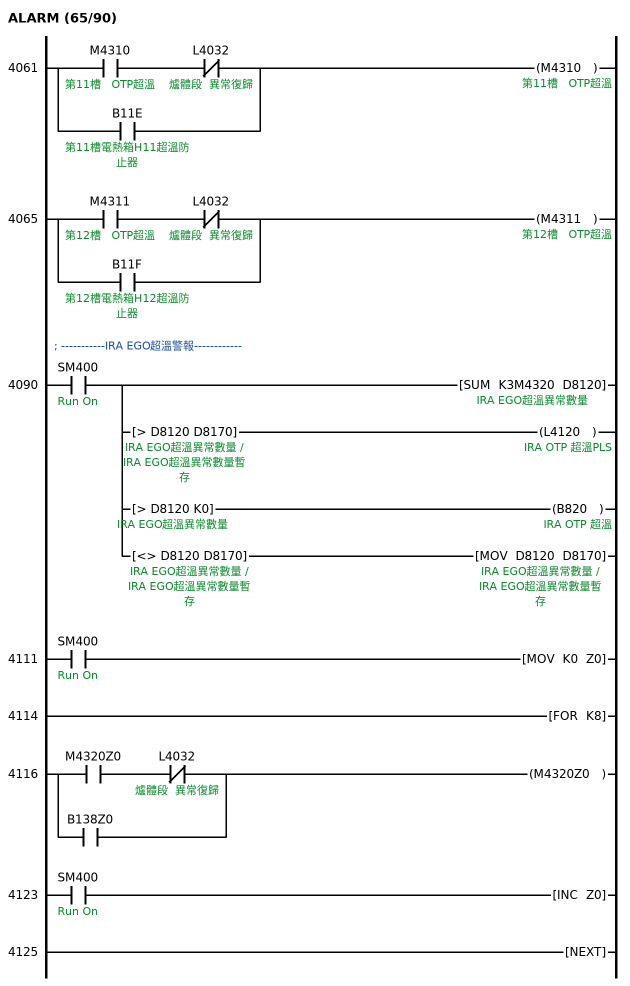
[picture p240: ladder of ALARM, rungs at steps 4061 to 4125]
4061  LD      M4310  ; 第11槽   OTP超溫
      ANI     L4032  ; 爐體段  異常復歸
      OR      B11E  ; 第11槽電熱箱H11超溫防止器
      OUT     M4310  ; 第11槽   OTP超溫
4065  LD      M4311  ; 第12槽   OTP超溫
      ANI     L4032  ; 爐體段  異常復歸
      OR      B11F  ; 第12槽電熱箱H12超溫防止器
      OUT     M4311  ; 第12槽   OTP超溫
; -----------IRA EGO超溫警報------------
4090  LD      SM400  ; Run On
      SUM     K3M4320 D8120  ; 第01槽  IRA OTP 超溫 / IRA EGO超溫異常數量
      MPS
      AND>    D8120 D8170  ; IRA EGO超溫異常數量 / IRA EGO超溫異常數量暫存
      OUT     L4120  ; IRA OTP 超溫PLS
      MRD
      AND>    D8120 K0  ; IRA EGO超溫異常數量
      OUT     B820  ; IRA OTP 超溫
      MPP
      AND<>   D8120 D8170  ; IRA EGO超溫異常數量 / IRA EGO超溫異常數量暫存
      MOV     D8120 D8170
4111  LD      SM400  ; Run On
      MOV     K0 Z0
4114  FOR     K8
4116  LD      M4320Z0
      ANI     L4032  ; 爐體段  異常復歸
      OR      B138Z0
      OUT     M4320Z0
4123  LD      SM400  ; Run On
      INC     Z0
4125  NEXT
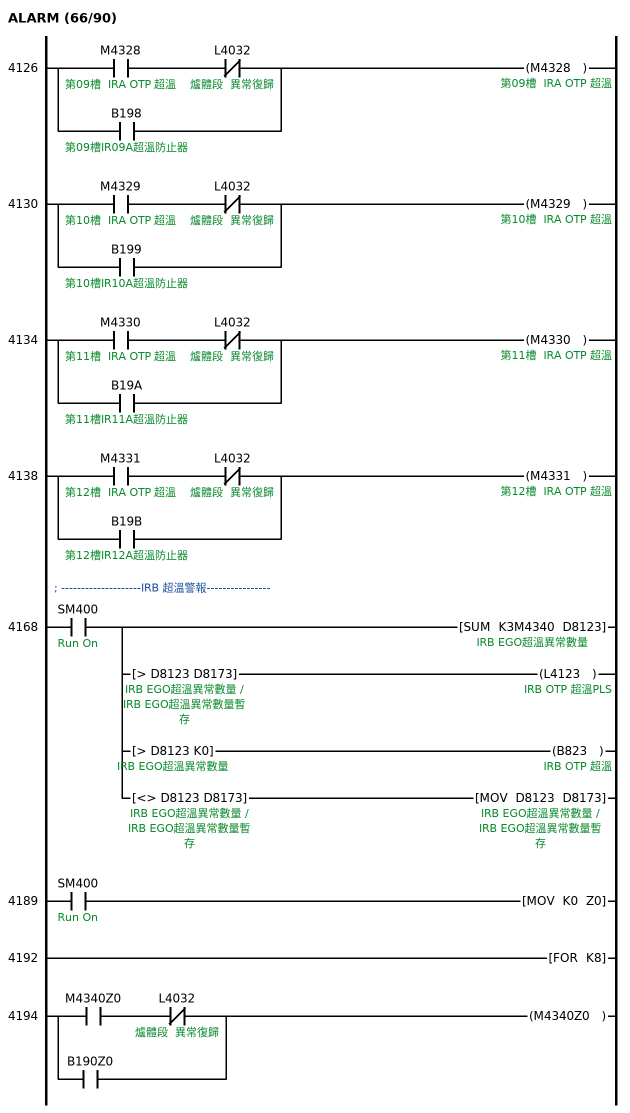
4126  LD      M4328  ; 第09槽  IRA OTP 超溫
      ANI     L4032  ; 爐體段  異常復歸
      OR      B198  ; 第09槽IR09A超溫防止器
      OUT     M4328  ; 第09槽  IRA OTP 超溫
4130  LD      M4329  ; 第10槽  IRA OTP 超溫
      ANI     L4032  ; 爐體段  異常復歸
      OR      B199  ; 第10槽IR10A超溫防止器
      OUT     M4329  ; 第10槽  IRA OTP 超溫
4134  LD      M4330  ; 第11槽  IRA OTP 超溫
      ANI     L4032  ; 爐體段  異常復歸
      OR      B19A  ; 第11槽IR11A超溫防止器
      OUT     M4330  ; 第11槽  IRA OTP 超溫
4138  LD      M4331  ; 第12槽  IRA OTP 超溫
      ANI     L4032  ; 爐體段  異常復歸
      OR      B19B  ; 第12槽IR12A超溫防止器
      OUT     M4331  ; 第12槽  IRA OTP 超溫
; --------------------IRB 超溫警報----------------
4168  LD      SM400  ; Run On
      SUM     K3M4340 D8123  ; 第01槽  IRB OTP 超溫 / IRB EGO超溫異常數量
      MPS
      AND>    D8123 D8173  ; IRB EGO超溫異常數量 / IRB EGO超溫異常數量暫存
      OUT     L4123  ; IRB OTP 超溫PLS
      MRD
      AND>    D8123 K0  ; IRB EGO超溫異常數量
      OUT     B823  ; IRB OTP 超溫
      MPP
      AND<>   D8123 D8173  ; IRB EGO超溫異常數量 / IRB EGO超溫異常數量暫存
      MOV     D8123 D8173
4189  LD      SM400  ; Run On
      MOV     K0 Z0
4192  FOR     K8
4194  LD      M4340Z0
      ANI     L4032  ; 爐體段  異常復歸
      OR      B190Z0
      OUT     M4340Z0
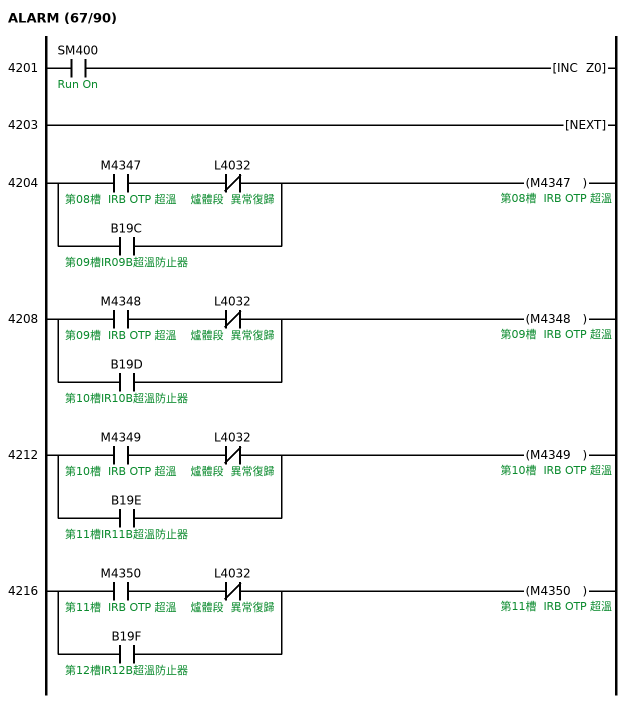
4201  LD      SM400  ; Run On
      INC     Z0
4203  NEXT
4204  LD      M4347  ; 第08槽  IRB OTP 超溫
      ANI     L4032  ; 爐體段  異常復歸
      OR      B19C  ; 第09槽IR09B超溫防止器
      OUT     M4347  ; 第08槽  IRB OTP 超溫
4208  LD      M4348  ; 第09槽  IRB OTP 超溫
      ANI     L4032  ; 爐體段  異常復歸
      OR      B19D  ; 第10槽IR10B超溫防止器
      OUT     M4348  ; 第09槽  IRB OTP 超溫
4212  LD      M4349  ; 第10槽  IRB OTP 超溫
      ANI     L4032  ; 爐體段  異常復歸
      OR      B19E  ; 第11槽IR11B超溫防止器
      OUT     M4349  ; 第10槽  IRB OTP 超溫
4216  LD      M4350  ; 第11槽  IRB OTP 超溫
      ANI     L4032  ; 爐體段  異常復歸
      OR      B19F  ; 第12槽IR12B超溫防止器
      OUT     M4350  ; 第11槽  IRB OTP 超溫
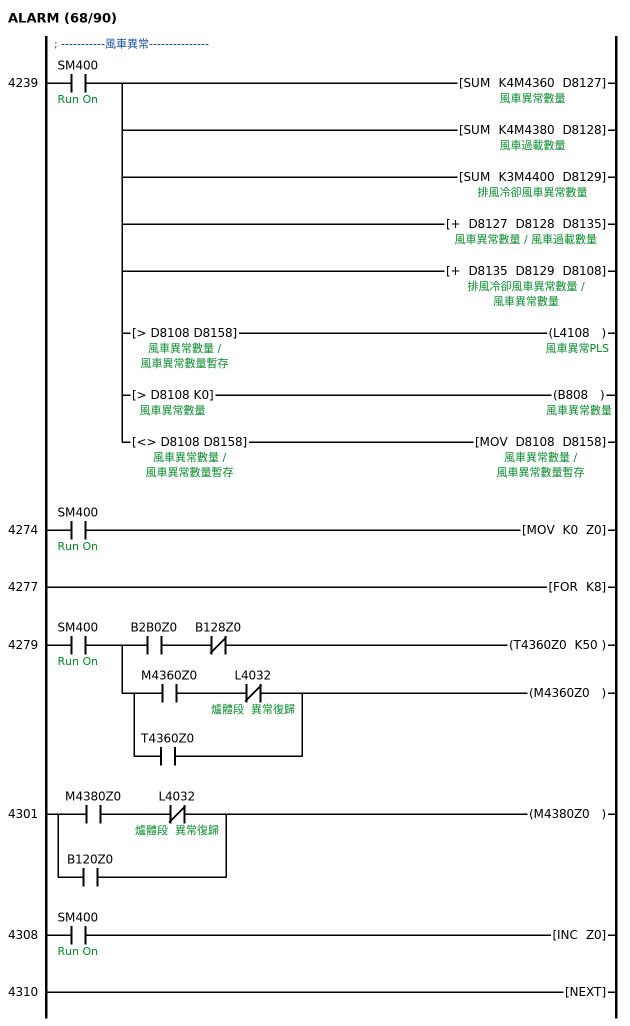
; -----------風車異常---------------
4239  LD      SM400  ; Run On
      SUM     K4M4360 D8127  ; 第01槽  風車馬達異常 / 風車異常數量
      SUM     K4M4380 D8128  ; 第01槽  風車馬達過載 / 風車過載數量
      SUM     K3M4400 D8129  ; 進料輸送排氣風車異常 / 排風冷卻風車異常數量
      +       D8127 D8128 D8135
      +       D8135 D8129 D8108  ; 風車異常數量
      MPS
      AND>    D8108 D8158  ; 風車異常數量 / 風車異常數量暫存
      OUT     L4108  ; 風車異常PLS
      MRD
      AND>    D8108 K0  ; 風車異常數量
      OUT     B808  ; 風車異常數量
      MPP
      AND<>   D8108 D8158  ; 風車異常數量 / 風車異常數量暫存
      MOV     D8108 D8158
4274  LD      SM400  ; Run On
      MOV     K0 Z0
4277  FOR     K8
4279  LD      SM400  ; Run On
      MPS
      AND     B2B0Z0
      ANI     B128Z0
      OUT     T4360Z0 K50
      MPP
      LD      M4360Z0
      ANI     L4032  ; 爐體段  異常復歸
      OR      T4360Z0
      ANB
      OUT     M4360Z0
4301  LD      M4380Z0
      ANI     L4032  ; 爐體段  異常復歸
      OR      B120Z0
      OUT     M4380Z0
4308  LD      SM400  ; Run On
      INC     Z0
4310  NEXT
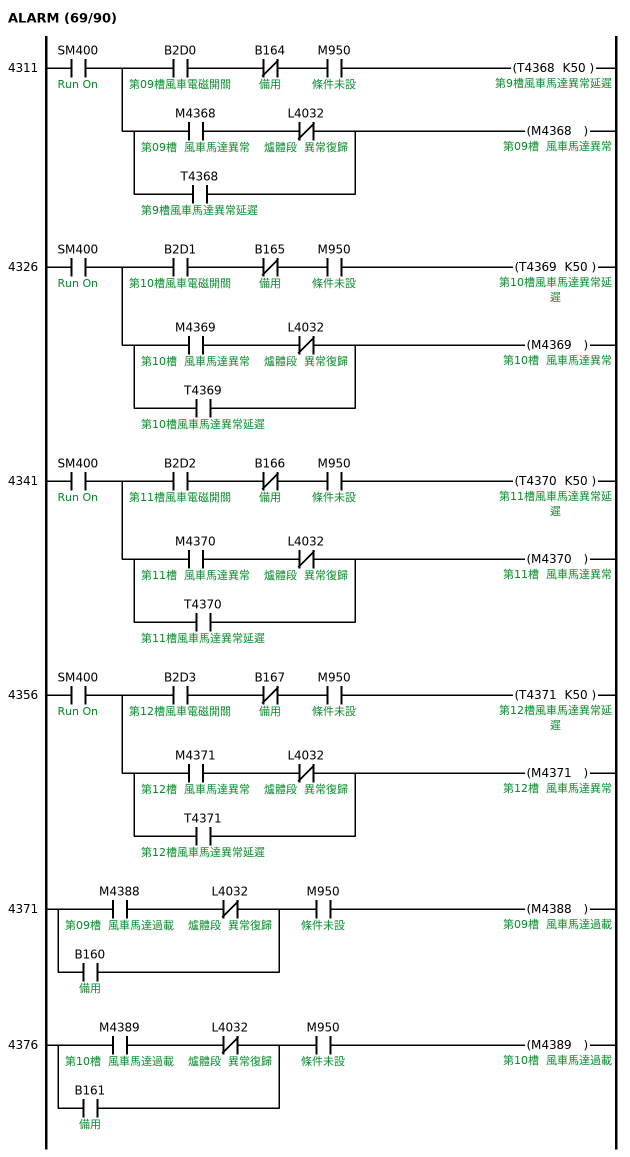
4311  LD      SM400  ; Run On
      MPS
      AND     B2D0  ; 第09槽風車電磁開關
      ANI     B164  ; 備用
      AND     M950  ; 條件未設
      OUT     T4368 K50  ; 第9槽風車馬達異常延遲
      MPP
      LD      M4368  ; 第09槽  風車馬達異常
      ANI     L4032  ; 爐體段  異常復歸
      OR      T4368  ; 第9槽風車馬達異常延遲
      ANB
      OUT     M4368  ; 第09槽  風車馬達異常
4326  LD      SM400  ; Run On
      MPS
      AND     B2D1  ; 第10槽風車電磁開關
      ANI     B165  ; 備用
      AND     M950  ; 條件未設
      OUT     T4369 K50  ; 第10槽風車馬達異常延遲
      MPP
      LD      M4369  ; 第10槽  風車馬達異常
      ANI     L4032  ; 爐體段  異常復歸
      OR      T4369  ; 第10槽風車馬達異常延遲
      ANB
      OUT     M4369  ; 第10槽  風車馬達異常
4341  LD      SM400  ; Run On
      MPS
      AND     B2D2  ; 第11槽風車電磁開關
      ANI     B166  ; 備用
      AND     M950  ; 條件未設
      OUT     T4370 K50  ; 第11槽風車馬達異常延遲
      MPP
      LD      M4370  ; 第11槽  風車馬達異常
      ANI     L4032  ; 爐體段  異常復歸
      OR      T4370  ; 第11槽風車馬達異常延遲
      ANB
      OUT     M4370  ; 第11槽  風車馬達異常
4356  LD      SM400  ; Run On
      MPS
      AND     B2D3  ; 第12槽風車電磁開關
      ANI     B167  ; 備用
      AND     M950  ; 條件未設
      OUT     T4371 K50  ; 第12槽風車馬達異常延遲
      MPP
      LD      M4371  ; 第12槽  風車馬達異常
      ANI     L4032  ; 爐體段  異常復歸
      OR      T4371  ; 第12槽風車馬達異常延遲
      ANB
      OUT     M4371  ; 第12槽  風車馬達異常
4371  LD      M4388  ; 第09槽  風車馬達過載
      ANI     L4032  ; 爐體段  異常復歸
      OR      B160  ; 備用
      AND     M950  ; 條件未設
      OUT     M4388  ; 第09槽  風車馬達過載
4376  LD      M4389  ; 第10槽  風車馬達過載
      ANI     L4032  ; 爐體段  異常復歸
      OR      B161  ; 備用
      AND     M950  ; 條件未設
      OUT     M4389  ; 第10槽  風車馬達過載
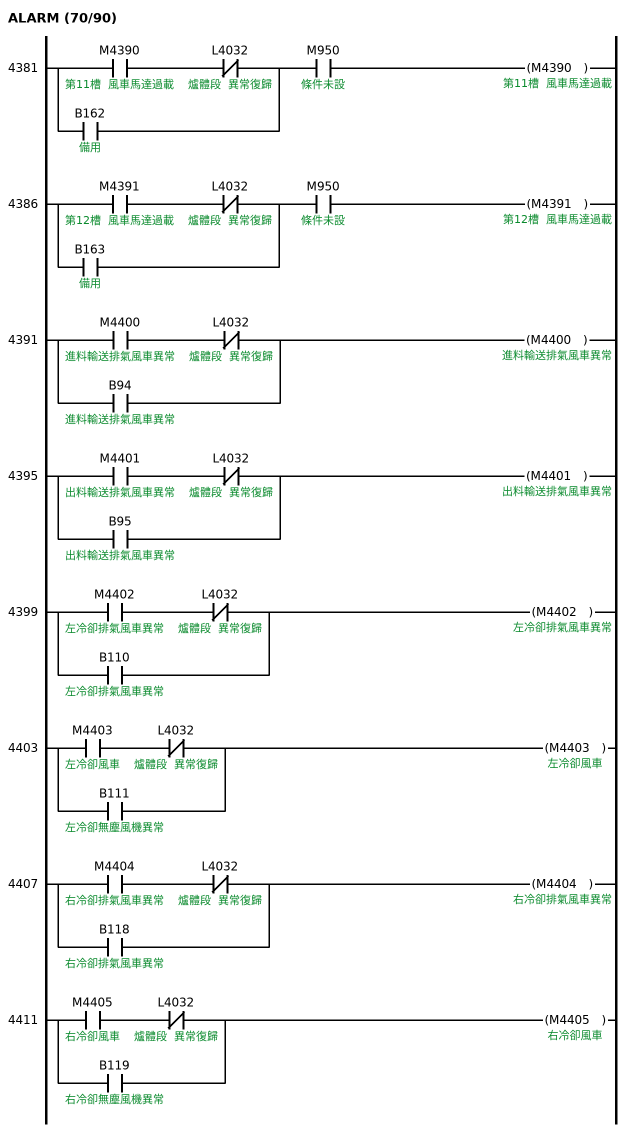
4381  LD      M4390  ; 第11槽  風車馬達過載
      ANI     L4032  ; 爐體段  異常復歸
      OR      B162  ; 備用
      AND     M950  ; 條件未設
      OUT     M4390  ; 第11槽  風車馬達過載
4386  LD      M4391  ; 第12槽  風車馬達過載
      ANI     L4032  ; 爐體段  異常復歸
      OR      B163  ; 備用
      AND     M950  ; 條件未設
      OUT     M4391  ; 第12槽  風車馬達過載
4391  LD      M4400  ; 進料輸送排氣風車異常
      ANI     L4032  ; 爐體段  異常復歸
      OR      B94  ; 進料輸送排氣風車異常
      OUT     M4400  ; 進料輸送排氣風車異常
4395  LD      M4401  ; 出料輸送排氣風車異常
      ANI     L4032  ; 爐體段  異常復歸
      OR      B95  ; 出料輸送排氣風車異常
      OUT     M4401  ; 出料輸送排氣風車異常
4399  LD      M4402  ; 左冷卻排氣風車異常
      ANI     L4032  ; 爐體段  異常復歸
      OR      B110  ; 左冷卻排氣風車異常
      OUT     M4402  ; 左冷卻排氣風車異常
4403  LD      M4403  ; 左冷卻風車
      ANI     L4032  ; 爐體段  異常復歸
      OR      B111  ; 左冷卻無塵風機異常
      OUT     M4403  ; 左冷卻風車
4407  LD      M4404  ; 右冷卻排氣風車異常
      ANI     L4032  ; 爐體段  異常復歸
      OR      B118  ; 右冷卻排氣風車異常
      OUT     M4404  ; 右冷卻排氣風車異常
4411  LD      M4405  ; 右冷卻風車
      ANI     L4032  ; 爐體段  異常復歸
      OR      B119  ; 右冷卻無塵風機異常
      OUT     M4405  ; 右冷卻風車
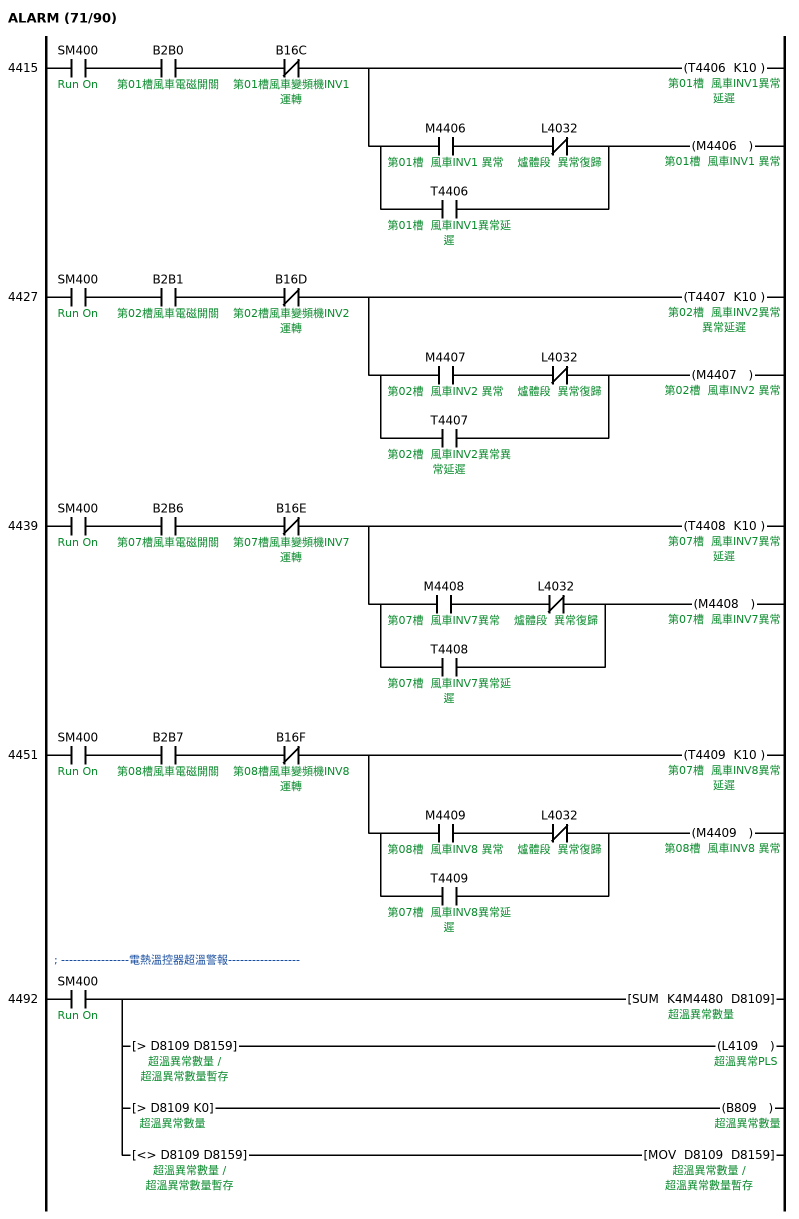
4415  LD      SM400  ; Run On
      AND     B2B0  ; 第01槽風車電磁開關
      ANI     B16C  ; 第01槽風車變頻機INV1運轉
      OUT     T4406 K10  ; 第01槽  風車INV1異常延遲
      LD      M4406  ; 第01槽  風車INV1 異常
      ANI     L4032  ; 爐體段  異常復歸
      OR      T4406  ; 第01槽  風車INV1異常延遲
      ANB
      OUT     M4406  ; 第01槽  風車INV1 異常
4427  LD      SM400  ; Run On
      AND     B2B1  ; 第02槽風車電磁開關
      ANI     B16D  ; 第02槽風車變頻機INV2運轉
      OUT     T4407 K10  ; 第02槽  風車INV2異常異常延遲
      LD      M4407  ; 第02槽  風車INV2 異常
      ANI     L4032  ; 爐體段  異常復歸
      OR      T4407  ; 第02槽  風車INV2異常異常延遲
      ANB
      OUT     M4407  ; 第02槽  風車INV2 異常
4439  LD      SM400  ; Run On
      AND     B2B6  ; 第07槽風車電磁開關
      ANI     B16E  ; 第07槽風車變頻機INV7運轉
      OUT     T4408 K10  ; 第07槽  風車INV7異常延遲
      LD      M4408  ; 第07槽  風車INV7異常
      ANI     L4032  ; 爐體段  異常復歸
      OR      T4408  ; 第07槽  風車INV7異常延遲
      ANB
      OUT     M4408  ; 第07槽  風車INV7異常
4451  LD      SM400  ; Run On
      AND     B2B7  ; 第08槽風車電磁開關
      ANI     B16F  ; 第08槽風車變頻機INV8運轉
      OUT     T4409 K10  ; 第07槽  風車INV8異常延遲
      LD      M4409  ; 第08槽  風車INV8 異常
      ANI     L4032  ; 爐體段  異常復歸
      OR      T4409  ; 第07槽  風車INV8異常延遲
      ANB
      OUT     M4409  ; 第08槽  風車INV8 異常
; -----------------電熱溫控器超溫警報------------------
4492  LD      SM400  ; Run On
      SUM     K4M4480 D8109  ; 第01槽 熱風超溫異常 / 超溫異常數量
      MPS
      AND>    D8109 D8159  ; 超溫異常數量 / 超溫異常數量暫存
      OUT     L4109  ; 超溫異常PLS
      MRD
      AND>    D8109 K0  ; 超溫異常數量
      OUT     B809  ; 超溫異常數量
      MPP
      AND<>   D8109 D8159  ; 超溫異常數量 / 超溫異常數量暫存
      MOV     D8109 D8159
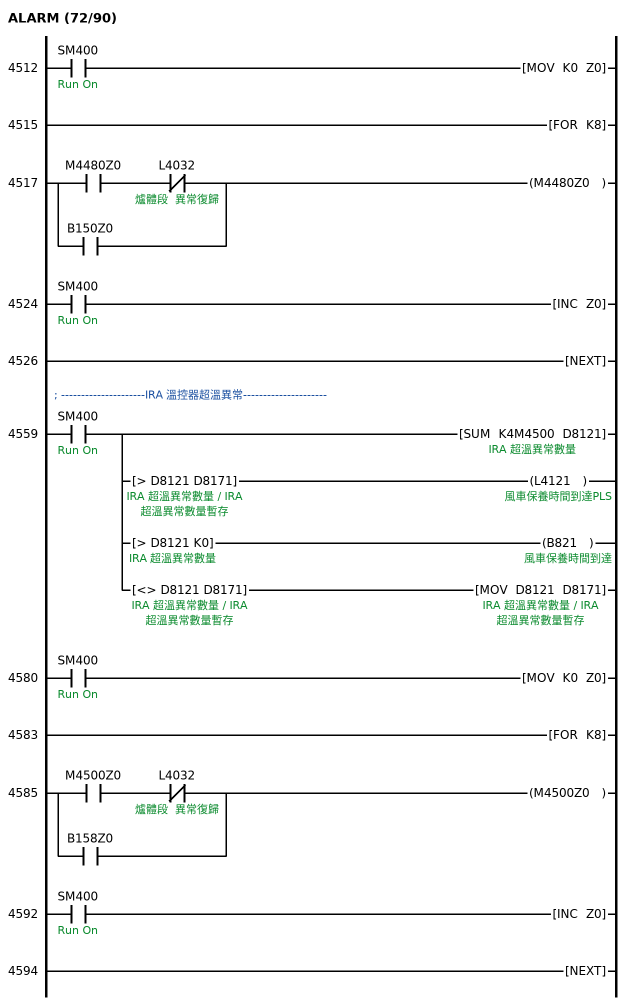
4512  LD      SM400  ; Run On
      MOV     K0 Z0
4515  FOR     K8
4517  LD      M4480Z0
      ANI     L4032  ; 爐體段  異常復歸
      OR      B150Z0
      OUT     M4480Z0
4524  LD      SM400  ; Run On
      INC     Z0
4526  NEXT
; ---------------------IRA 溫控器超溫異常---------------------
4559  LD      SM400  ; Run On
      SUM     K4M4500 D8121  ; 第1槽 IRA 超溫異常 / IRA 超溫異常數量
      MPS
      AND>    D8121 D8171  ; IRA 超溫異常數量 / IRA 超溫異常數量暫存
      OUT     L4121  ; 風車保養時間到達PLS
      MRD
      AND>    D8121 K0  ; IRA 超溫異常數量
      OUT     B821  ; 風車保養時間到達
      MPP
      AND<>   D8121 D8171  ; IRA 超溫異常數量 / IRA 超溫異常數量暫存
      MOV     D8121 D8171
4580  LD      SM400  ; Run On
      MOV     K0 Z0
4583  FOR     K8
4585  LD      M4500Z0
      ANI     L4032  ; 爐體段  異常復歸
      OR      B158Z0
      OUT     M4500Z0
4592  LD      SM400  ; Run On
      INC     Z0
4594  NEXT
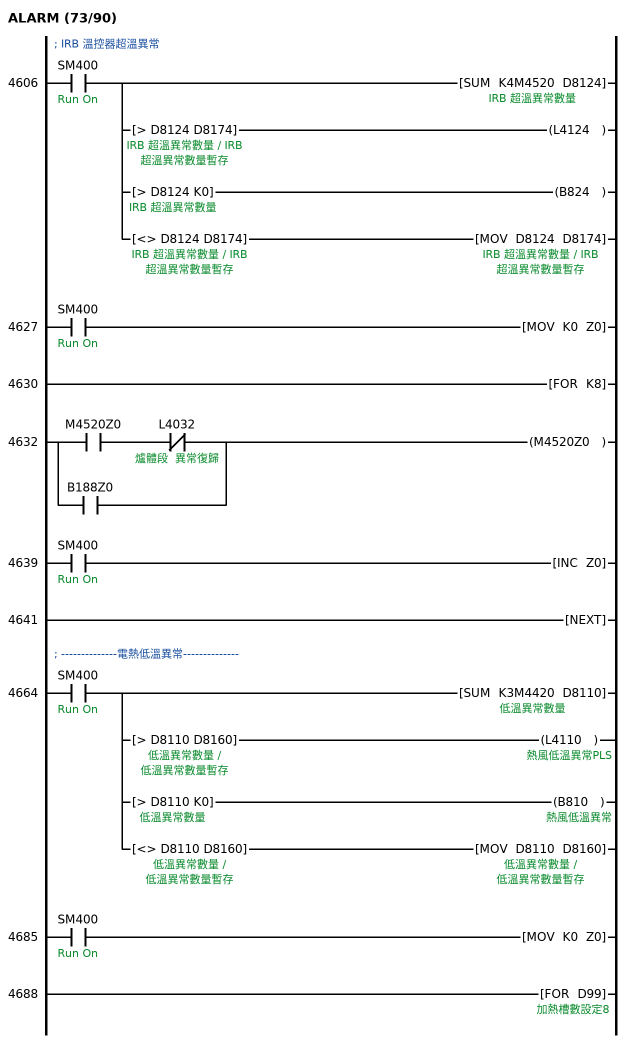
; IRB 溫控器超溫異常
4606  LD      SM400  ; Run On
      SUM     K4M4520 D8124  ; 第1槽 IRB 超溫異常 / IRB 超溫異常數量
      MPS
      AND>    D8124 D8174  ; IRB 超溫異常數量 / IRB 超溫異常數量暫存
      OUT     L4124
      MRD
      AND>    D8124 K0  ; IRB 超溫異常數量
      OUT     B824
      MPP
      AND<>   D8124 D8174  ; IRB 超溫異常數量 / IRB 超溫異常數量暫存
      MOV     D8124 D8174
4627  LD      SM400  ; Run On
      MOV     K0 Z0
4630  FOR     K8
4632  LD      M4520Z0
      ANI     L4032  ; 爐體段  異常復歸
      OR      B188Z0
      OUT     M4520Z0
4639  LD      SM400  ; Run On
      INC     Z0
4641  NEXT
; --------------電熱低溫異常--------------
4664  LD      SM400  ; Run On
      SUM     K3M4420 D8110  ; 第01槽 熱風低溫異常 / 低溫異常數量
      MPS
      AND>    D8110 D8160  ; 低溫異常數量 / 低溫異常數量暫存
      OUT     L4110  ; 熱風低溫異常PLS
      MRD
      AND>    D8110 K0  ; 低溫異常數量
      OUT     B810  ; 熱風低溫異常
      MPP
      AND<>   D8110 D8160  ; 低溫異常數量 / 低溫異常數量暫存
      MOV     D8110 D8160
4685  LD      SM400  ; Run On
      MOV     K0 Z0
4688  FOR     D99  ; 加熱槽數設定8
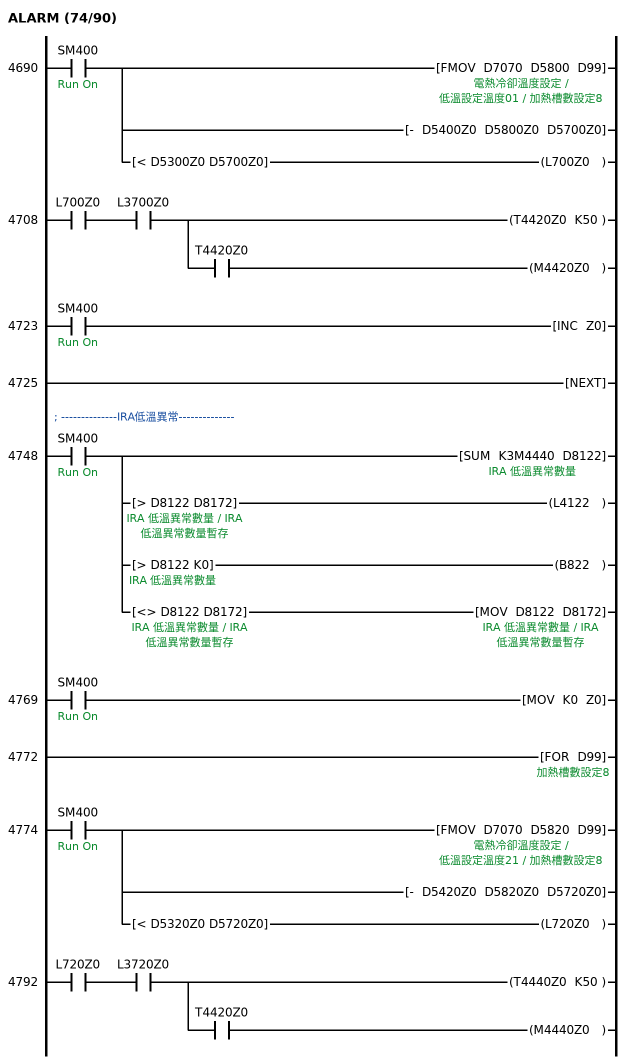
4690  LD      SM400  ; Run On
      FMOV    D7070 D5800 D99  ; 電熱冷卻溫度設定 / 低溫設定溫度01
      -       D5400Z0 D5800Z0 D5700Z0
      AND<    D5300Z0 D5700Z0
      OUT     L700Z0
4708  LD      L700Z0
      AND     L3700Z0
      OUT     T4420Z0 K50
      AND     T4420Z0
      OUT     M4420Z0
4723  LD      SM400  ; Run On
      INC     Z0
4725  NEXT
; --------------IRA低溫異常--------------
4748  LD      SM400  ; Run On
      SUM     K3M4440 D8122  ; 第01槽 IRA 低溫異常 / IRA 低溫異常數量
      MPS
      AND>    D8122 D8172  ; IRA 低溫異常數量 / IRA 低溫異常數量暫存
      OUT     L4122
      MRD
      AND>    D8122 K0  ; IRA 低溫異常數量
      OUT     B822
      MPP
      AND<>   D8122 D8172  ; IRA 低溫異常數量 / IRA 低溫異常數量暫存
      MOV     D8122 D8172
4769  LD      SM400  ; Run On
      MOV     K0 Z0
4772  FOR     D99
4774  LD      SM400  ; Run On
      FMOV    D7070 D5820 D99  ; 低溫設定溫度21
      -       D5420Z0 D5820Z0 D5720Z0
      AND<    D5320Z0 D5720Z0
      OUT     L720Z0
4792  LD      L720Z0
      AND     L3720Z0
      OUT     T4440Z0 K50
      AND     T4420Z0
      OUT     M4440Z0
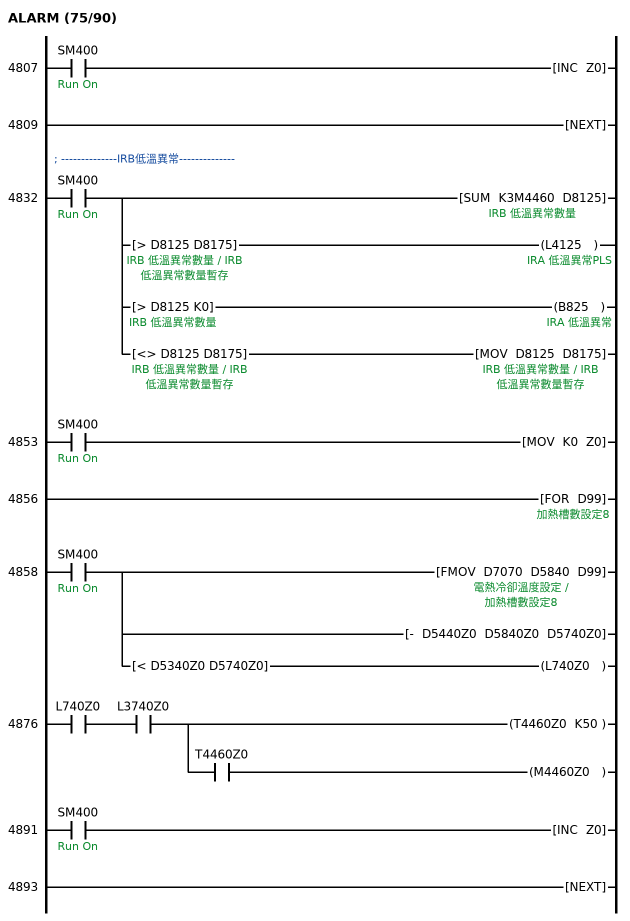
4807  LD      SM400  ; Run On
      INC     Z0
4809  NEXT
; --------------IRB低溫異常--------------
4832  LD      SM400  ; Run On
      SUM     K3M4460 D8125  ; 第01槽 IRB 低溫異常 / IRB 低溫異常數量
      MPS
      AND>    D8125 D8175  ; IRB 低溫異常數量 / IRB 低溫異常數量暫存
      OUT     L4125  ; IRA 低溫異常PLS
      MRD
      AND>    D8125 K0  ; IRB 低溫異常數量
      OUT     B825  ; IRA 低溫異常
      MPP
      AND<>   D8125 D8175  ; IRB 低溫異常數量 / IRB 低溫異常數量暫存
      MOV     D8125 D8175
4853  LD      SM400  ; Run On
      MOV     K0 Z0
4856  FOR     D99
4858  LD      SM400  ; Run On
      FMOV    D7070 D5840 D99
      -       D5440Z0 D5840Z0 D5740Z0
      AND<    D5340Z0 D5740Z0
      OUT     L740Z0
4876  LD      L740Z0
      AND     L3740Z0
      OUT     T4460Z0 K50
      AND     T4460Z0
      OUT     M4460Z0
4891  LD      SM400  ; Run On
      INC     Z0
4893  NEXT
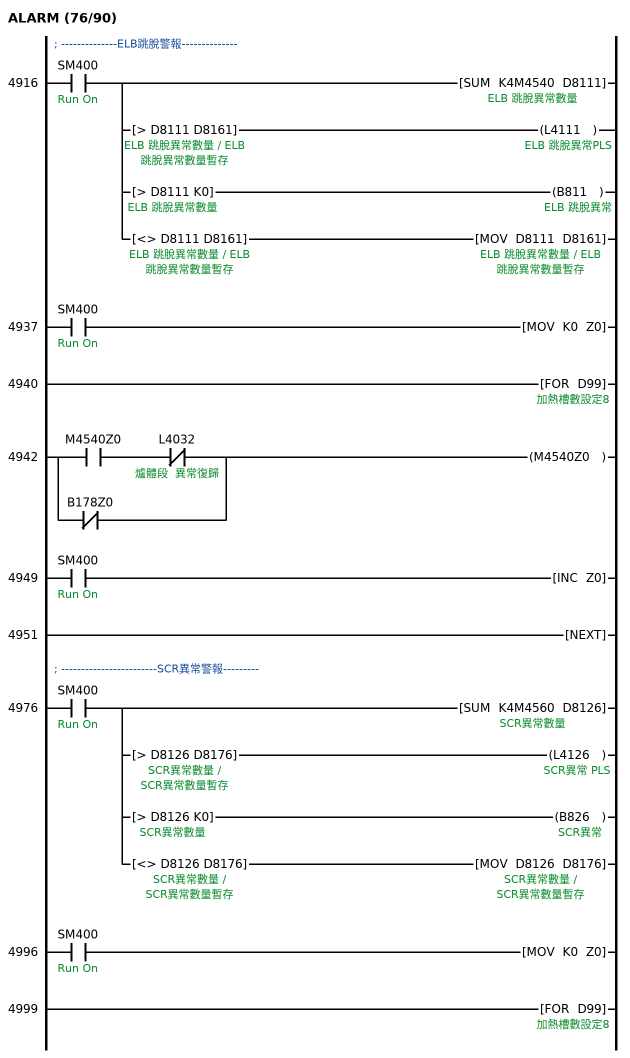
; --------------ELB跳脫警報--------------
4916  LD      SM400  ; Run On
      SUM     K4M4540 D8111  ; 第01槽  分路開關跳脫異常 / ELB 跳脫異常數量
      MPS
      AND>    D8111 D8161  ; ELB 跳脫異常數量 / ELB 跳脫異常數量暫存
      OUT     L4111  ; ELB 跳脫異常PLS
      MRD
      AND>    D8111 K0  ; ELB 跳脫異常數量
      OUT     B811  ; ELB 跳脫異常
      MPP
      AND<>   D8111 D8161  ; ELB 跳脫異常數量 / ELB 跳脫異常數量暫存
      MOV     D8111 D8161
4937  LD      SM400  ; Run On
      MOV     K0 Z0
4940  FOR     D99
4942  LD      M4540Z0
      ANI     L4032  ; 爐體段  異常復歸
      ORI     B178Z0
      OUT     M4540Z0
4949  LD      SM400  ; Run On
      INC     Z0
4951  NEXT
; ------------------------SCR異常警報---------
4976  LD      SM400  ; Run On
      SUM     K4M4560 D8126  ; 第01槽  SCR異常 / SCR異常數量
      MPS
      AND>    D8126 D8176  ; SCR異常數量 / SCR異常數量暫存
      OUT     L4126  ; SCR異常 PLS
      MRD
      AND>    D8126 K0  ; SCR異常數量
      OUT     B826  ; SCR異常
      MPP
      AND<>   D8126 D8176  ; SCR異常數量 / SCR異常數量暫存
      MOV     D8126 D8176
4996  LD      SM400  ; Run On
      MOV     K0 Z0
4999  FOR     D99
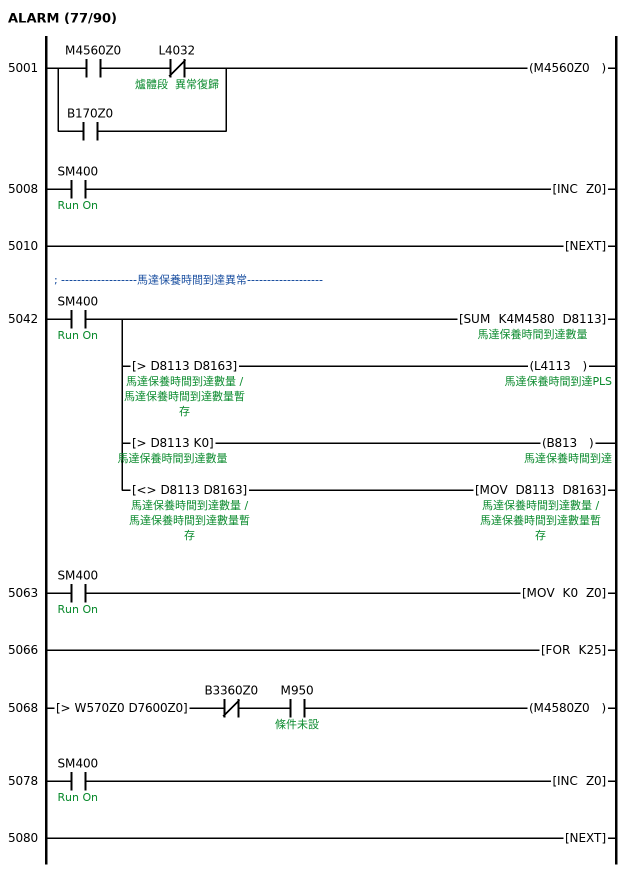
5001  LD      M4560Z0
      ANI     L4032  ; 爐體段  異常復歸
      OR      B170Z0
      OUT     M4560Z0
5008  LD      SM400  ; Run On
      INC     Z0
5010  NEXT
; -------------------馬達保養時間到達異常-------------------
5042  LD      SM400  ; Run On
      SUM     K4M4580 D8113  ; 馬達保養時間到達數量
      MPS
      AND>    D8113 D8163  ; 馬達保養時間到達數量 / 馬達保養時間到達數量暫存
      OUT     L4113  ; 馬達保養時間到達PLS
      MRD
      AND>    D8113 K0  ; 馬達保養時間到達數量
      OUT     B813  ; 馬達保養時間到達
      MPP
      AND<>   D8113 D8163  ; 馬達保養時間到達數量 / 馬達保養時間到達數量暫存
      MOV     D8113 D8163
5063  LD      SM400  ; Run On
      MOV     K0 Z0
5066  FOR     K25
5068  LD>     W570Z0 D7600Z0
      ANI     B3360Z0
      AND     M950  ; 條件未設
      OUT     M4580Z0
5078  LD      SM400  ; Run On
      INC     Z0
5080  NEXT
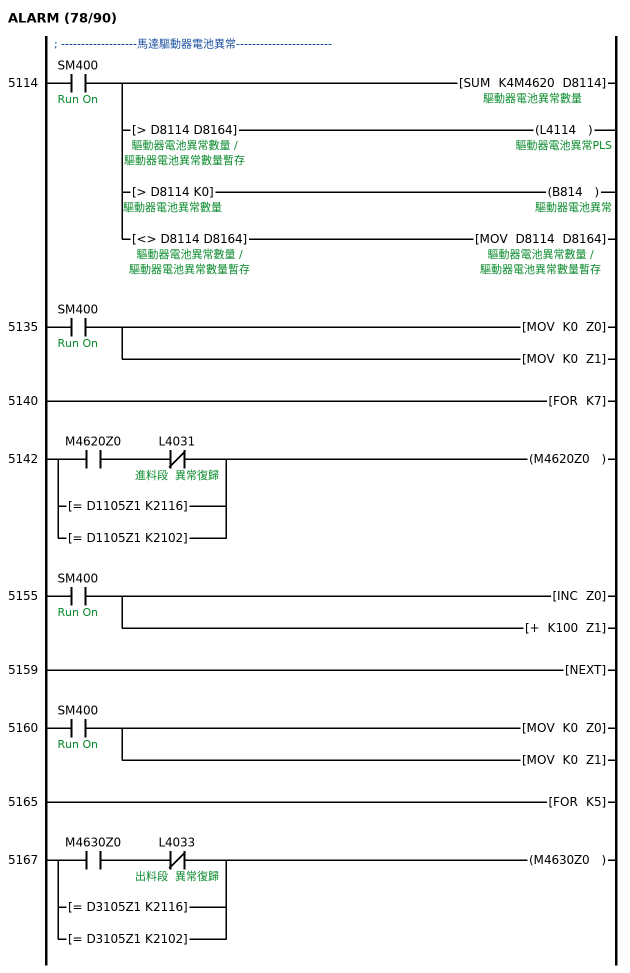
; -------------------馬達驅動器電池異常------------------------
5114  LD      SM400  ; Run On
      SUM     K4M4620 D8114  ; 進料整板驅動器電池異常 / 驅動器電池異常數量
      MPS
      AND>    D8114 D8164  ; 驅動器電池異常數量 / 驅動器電池異常數量暫存
      OUT     L4114  ; 驅動器電池異常PLS
      MRD
      AND>    D8114 K0  ; 驅動器電池異常數量
      OUT     B814  ; 驅動器電池異常
      MPP
      AND<>   D8114 D8164  ; 驅動器電池異常數量 / 驅動器電池異常數量暫存
      MOV     D8114 D8164
5135  LD      SM400  ; Run On
      MOV     K0 Z0
      MOV     K0 Z1
5140  FOR     K7
5142  LD      M4620Z0
      ANI     L4031  ; 進料段  異常復歸
      OR=     D1105Z1 K2116
      OR=     D1105Z1 K2102
      OUT     M4620Z0
5155  LD      SM400  ; Run On
      INC     Z0
      +       K100 Z1
5159  NEXT
5160  LD      SM400  ; Run On
      MOV     K0 Z0
      MOV     K0 Z1
5165  FOR     K5
5167  LD      M4630Z0
      ANI     L4033  ; 出料段  異常復歸
      OR=     D3105Z1 K2116
      OR=     D3105Z1 K2102
      OUT     M4630Z0
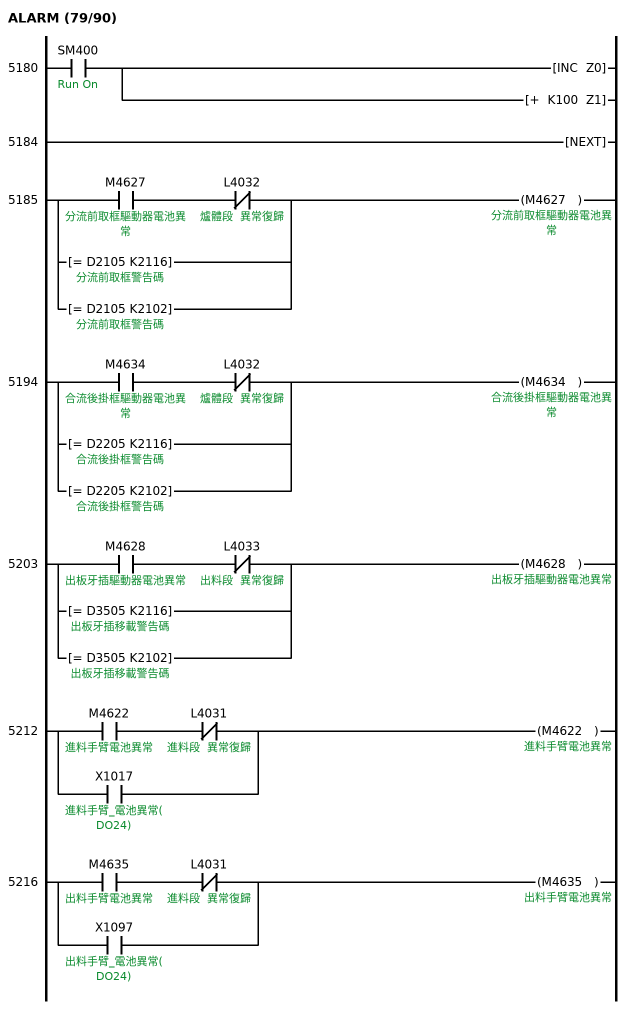
5180  LD      SM400  ; Run On
      INC     Z0
      +       K100 Z1
5184  NEXT
5185  LD      M4627  ; 分流前取框驅動器電池異常
      ANI     L4032  ; 爐體段  異常復歸
      OR=     D2105 K2116  ; 分流前取框警告碼
      OR=     D2105 K2102  ; 分流前取框警告碼
      OUT     M4627  ; 分流前取框驅動器電池異常
5194  LD      M4634  ; 合流後掛框驅動器電池異常
      ANI     L4032  ; 爐體段  異常復歸
      OR=     D2205 K2116  ; 合流後掛框警告碼
      OR=     D2205 K2102  ; 合流後掛框警告碼
      OUT     M4634  ; 合流後掛框驅動器電池異常
5203  LD      M4628  ; 出板牙插驅動器電池異常
      ANI     L4033  ; 出料段  異常復歸
      OR=     D3505 K2116  ; 出板牙插移載警告碼
      OR=     D3505 K2102  ; 出板牙插移載警告碼
      OUT     M4628  ; 出板牙插驅動器電池異常
5212  LD      M4622  ; 進料手臂電池異常
      ANI     L4031  ; 進料段  異常復歸
      OR      X1017  ; 進料手臂_電池異常(DO24)
      OUT     M4622  ; 進料手臂電池異常
5216  LD      M4635  ; 出料手臂電池異常
      ANI     L4031  ; 進料段  異常復歸
      OR      X1097  ; 出料手臂_電池異常(DO24)
      OUT     M4635  ; 出料手臂電池異常
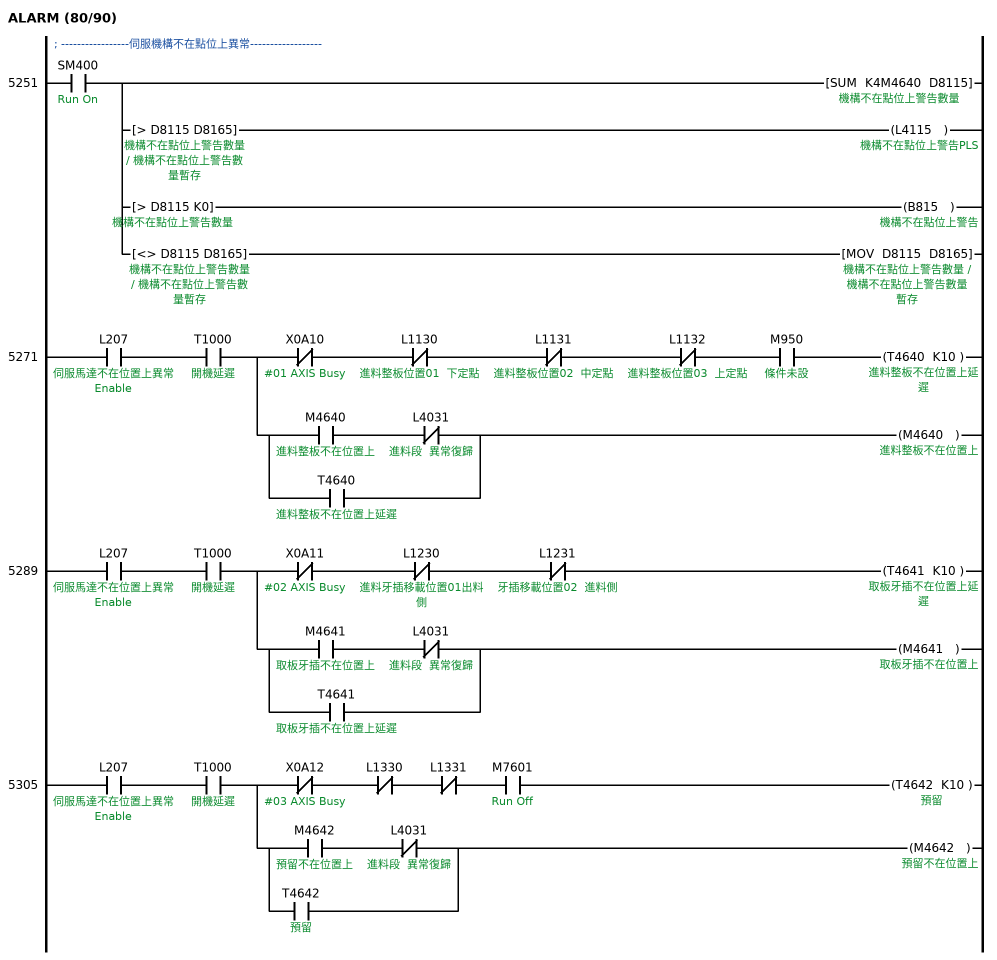
; -----------------伺服機構不在點位上異常------------------
5251  LD      SM400  ; Run On
      SUM     K4M4640 D8115  ; 進料整板不在位置上 / 機構不在點位上警告數量
      MPS
      AND>    D8115 D8165  ; 機構不在點位上警告數量 / 機構不在點位上警告數量暫存
      OUT     L4115  ; 機構不在點位上警告PLS
      MRD
      AND>    D8115 K0  ; 機構不在點位上警告數量
      OUT     B815  ; 機構不在點位上警告
      MPP
      AND<>   D8115 D8165  ; 機構不在點位上警告數量 / 機構不在點位上警告數量暫存
      MOV     D8115 D8165
5271  LD      L207  ; 伺服馬達不在位置上異常  Enable
      AND     T1000  ; 開機延遲
      MPS
      ANI     X0A10  ; #01 AXIS Busy
      ANI     L1130  ; 進料整板位置01  下定點
      ANI     L1131  ; 進料整板位置02  中定點
      ANI     L1132  ; 進料整板位置03  上定點
      AND     M950  ; 條件未設
      OUT     T4640 K10  ; 進料整板不在位置上延遲
      MPP
      LD      M4640  ; 進料整板不在位置上
      ANI     L4031  ; 進料段  異常復歸
      OR      T4640  ; 進料整板不在位置上延遲
      ANB
      OUT     M4640  ; 進料整板不在位置上
5289  LD      L207  ; 伺服馬達不在位置上異常  Enable
      AND     T1000  ; 開機延遲
      MPS
      ANI     X0A11  ; #02 AXIS Busy
      ANI     L1230  ; 進料牙插移載位置01出料側
      ANI     L1231  ; 牙插移載位置02  進料側
      OUT     T4641 K10  ; 取板牙插不在位置上延遲
      MPP
      LD      M4641  ; 取板牙插不在位置上
      ANI     L4031  ; 進料段  異常復歸
      OR      T4641  ; 取板牙插不在位置上延遲
      ANB
      OUT     M4641  ; 取板牙插不在位置上
5305  LD      L207  ; 伺服馬達不在位置上異常  Enable
      AND     T1000  ; 開機延遲
      MPS
      ANI     X0A12  ; #03 AXIS Busy
      ANI     L1330
      ANI     L1331
      AND     M7601  ; Run Off
      OUT     T4642 K10  ; 預留
      MPP
      LD      M4642  ; 預留不在位置上
      ANI     L4031  ; 進料段  異常復歸
      OR      T4642  ; 預留
      ANB
      OUT     M4642  ; 預留不在位置上
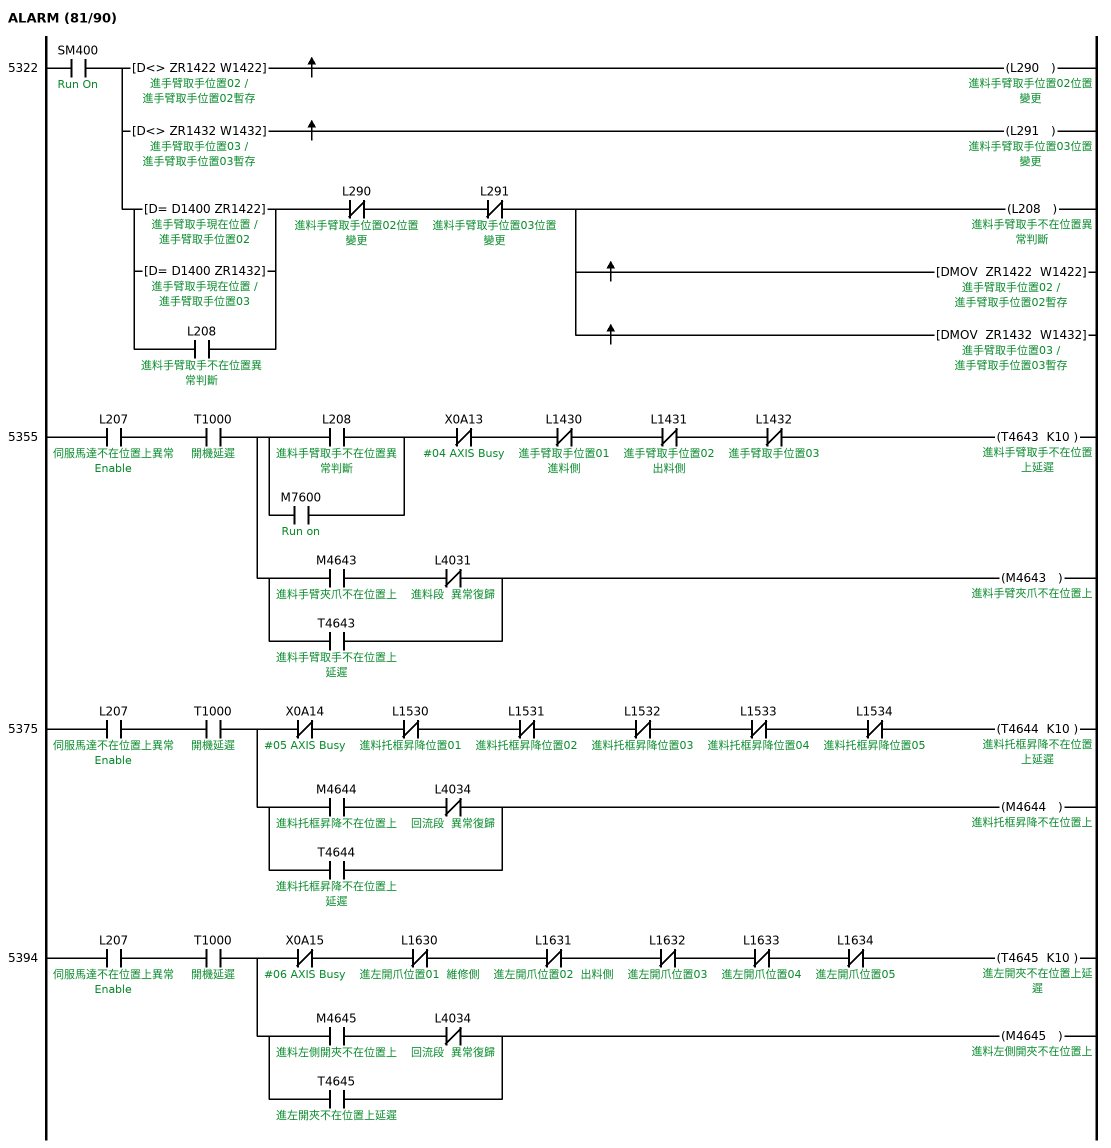
5322  LD      SM400  ; Run On
      MPS
      ANDD<>  ZR1422 W1422  ; 進手臂取手位置02 / 進手臂取手位置02暫存
      MEP
      OUT     L290  ; 進料手臂取手位置02位置變更
      MRD
      ANDD<>  ZR1432 W1432  ; 進手臂取手位置03 / 進手臂取手位置03暫存
      MEP
      OUT     L291  ; 進料手臂取手位置03位置變更
      MPP
      LDD=    D1400 ZR1422  ; 進手臂取手現在位置 / 進手臂取手位置02
      ORD=    D1400 ZR1432  ; 進手臂取手現在位置 / 進手臂取手位置03
      OR      L208  ; 進料手臂取手不在位置異常判斷
      ANB
      ANI     L290  ; 進料手臂取手位置02位置變更
      ANI     L291  ; 進料手臂取手位置03位置變更
      OUT     L208  ; 進料手臂取手不在位置異常判斷
      MPS
      MEP
      DMOV    ZR1422 W1422
      MPP
      MEP
      DMOV    ZR1432 W1432
5355  LD      L207  ; 伺服馬達不在位置上異常  Enable
      AND     T1000  ; 開機延遲
      MPS
      LD      L208  ; 進料手臂取手不在位置異常判斷
      OR      M7600  ; Run on
      ANB
      ANI     X0A13  ; #04 AXIS Busy
      ANI     L1430  ; 進手臂取手位置01  進料側
      ANI     L1431  ; 進手臂取手位置02  出料側
      ANI     L1432  ; 進手臂取手位置03
      OUT     T4643 K10  ; 進料手臂取手不在位置上延遲
      MPP
      LD      M4643  ; 進料手臂夾爪不在位置上
      ANI     L4031  ; 進料段  異常復歸
      OR      T4643  ; 進料手臂取手不在位置上延遲
      ANB
      OUT     M4643  ; 進料手臂夾爪不在位置上
5375  LD      L207  ; 伺服馬達不在位置上異常  Enable
      AND     T1000  ; 開機延遲
      MPS
      ANI     X0A14  ; #05 AXIS Busy
      ANI     L1530  ; 進料托框昇降位置01
      ANI     L1531  ; 進料托框昇降位置02
      ANI     L1532  ; 進料托框昇降位置03
      ANI     L1533  ; 進料托框昇降位置04
      ANI     L1534  ; 進料托框昇降位置05
      OUT     T4644 K10  ; 進料托框昇降不在位置上延遲
      MPP
      LD      M4644  ; 進料托框昇降不在位置上
      ANI     L4034  ; 回流段  異常復歸
      OR      T4644  ; 進料托框昇降不在位置上延遲
      ANB
      OUT     M4644  ; 進料托框昇降不在位置上
5394  LD      L207  ; 伺服馬達不在位置上異常  Enable
      AND     T1000  ; 開機延遲
      MPS
      ANI     X0A15  ; #06 AXIS Busy
      ANI     L1630  ; 進左開爪位置01  維修側
      ANI     L1631  ; 進左開爪位置02  出料側
      ANI     L1632  ; 進左開爪位置03
      ANI     L1633  ; 進左開爪位置04
      ANI     L1634  ; 進左開爪位置05
      OUT     T4645 K10  ; 進左開夾不在位置上延遲
      MPP
      LD      M4645  ; 進料左側開夾不在位置上
      ANI     L4034  ; 回流段  異常復歸
      OR      T4645  ; 進左開夾不在位置上延遲
      ANB
      OUT     M4645  ; 進料左側開夾不在位置上
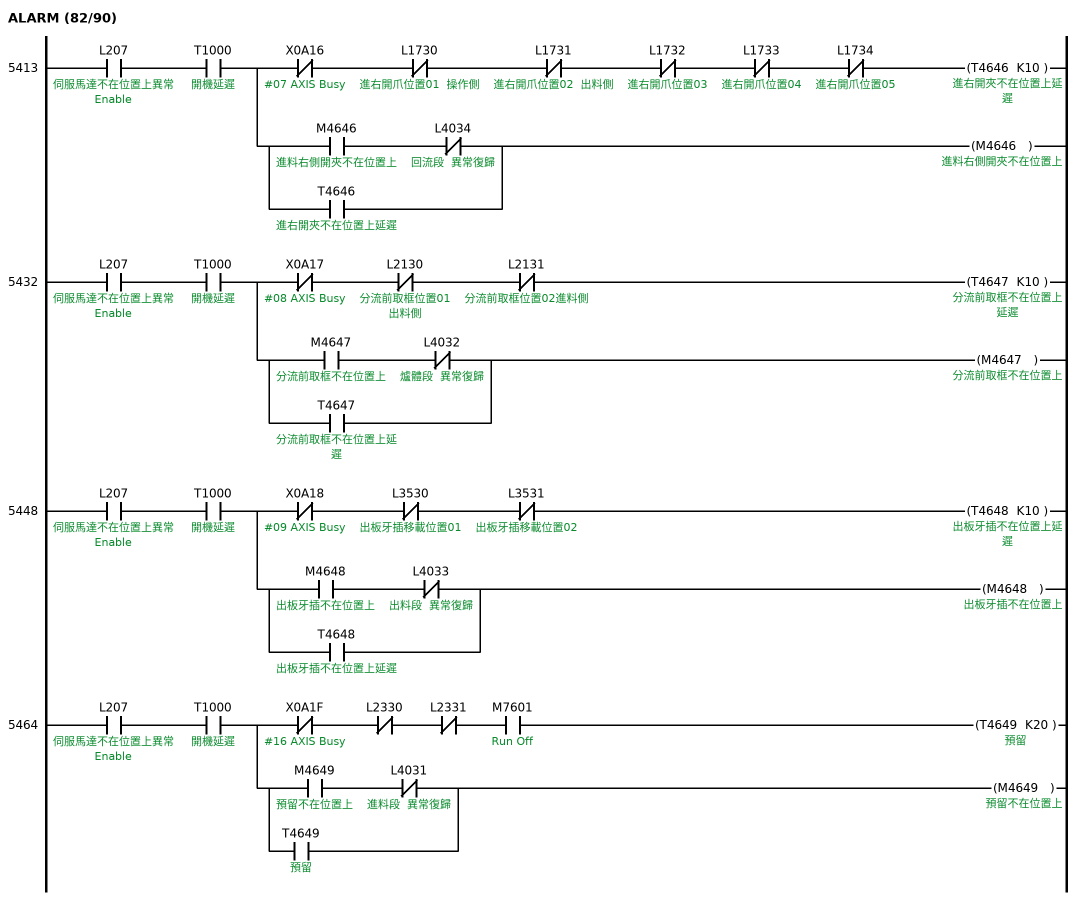
5413  LD      L207  ; 伺服馬達不在位置上異常  Enable
      AND     T1000  ; 開機延遲
      MPS
      ANI     X0A16  ; #07 AXIS Busy
      ANI     L1730  ; 進右開爪位置01  操作側
      ANI     L1731  ; 進右開爪位置02  出料側
      ANI     L1732  ; 進右開爪位置03
      ANI     L1733  ; 進右開爪位置04
      ANI     L1734  ; 進右開爪位置05
      OUT     T4646 K10  ; 進右開夾不在位置上延遲
      MPP
      LD      M4646  ; 進料右側開夾不在位置上
      ANI     L4034  ; 回流段  異常復歸
      OR      T4646  ; 進右開夾不在位置上延遲
      ANB
      OUT     M4646  ; 進料右側開夾不在位置上
5432  LD      L207  ; 伺服馬達不在位置上異常  Enable
      AND     T1000  ; 開機延遲
      MPS
      ANI     X0A17  ; #08 AXIS Busy
      ANI     L2130  ; 分流前取框位置01  出料側
      ANI     L2131  ; 分流前取框位置02進料側
      OUT     T4647 K10  ; 分流前取框不在位置上延遲
      MPP
      LD      M4647  ; 分流前取框不在位置上
      ANI     L4032  ; 爐體段  異常復歸
      OR      T4647  ; 分流前取框不在位置上延遲
      ANB
      OUT     M4647  ; 分流前取框不在位置上
5448  LD      L207  ; 伺服馬達不在位置上異常  Enable
      AND     T1000  ; 開機延遲
      MPS
      ANI     X0A18  ; #09 AXIS Busy
      ANI     L3530  ; 出板牙插移載位置01
      ANI     L3531  ; 出板牙插移載位置02
      OUT     T4648 K10  ; 出板牙插不在位置上延遲
      MPP
      LD      M4648  ; 出板牙插不在位置上
      ANI     L4033  ; 出料段  異常復歸
      OR      T4648  ; 出板牙插不在位置上延遲
      ANB
      OUT     M4648  ; 出板牙插不在位置上
5464  LD      L207  ; 伺服馬達不在位置上異常  Enable
      AND     T1000  ; 開機延遲
      MPS
      ANI     X0A1F  ; #16 AXIS Busy
      ANI     L2330
      ANI     L2331
      AND     M7601  ; Run Off
      OUT     T4649 K20  ; 預留
      MPP
      LD      M4649  ; 預留不在位置上
      ANI     L4031  ; 進料段  異常復歸
      OR      T4649  ; 預留
      ANB
      OUT     M4649  ; 預留不在位置上
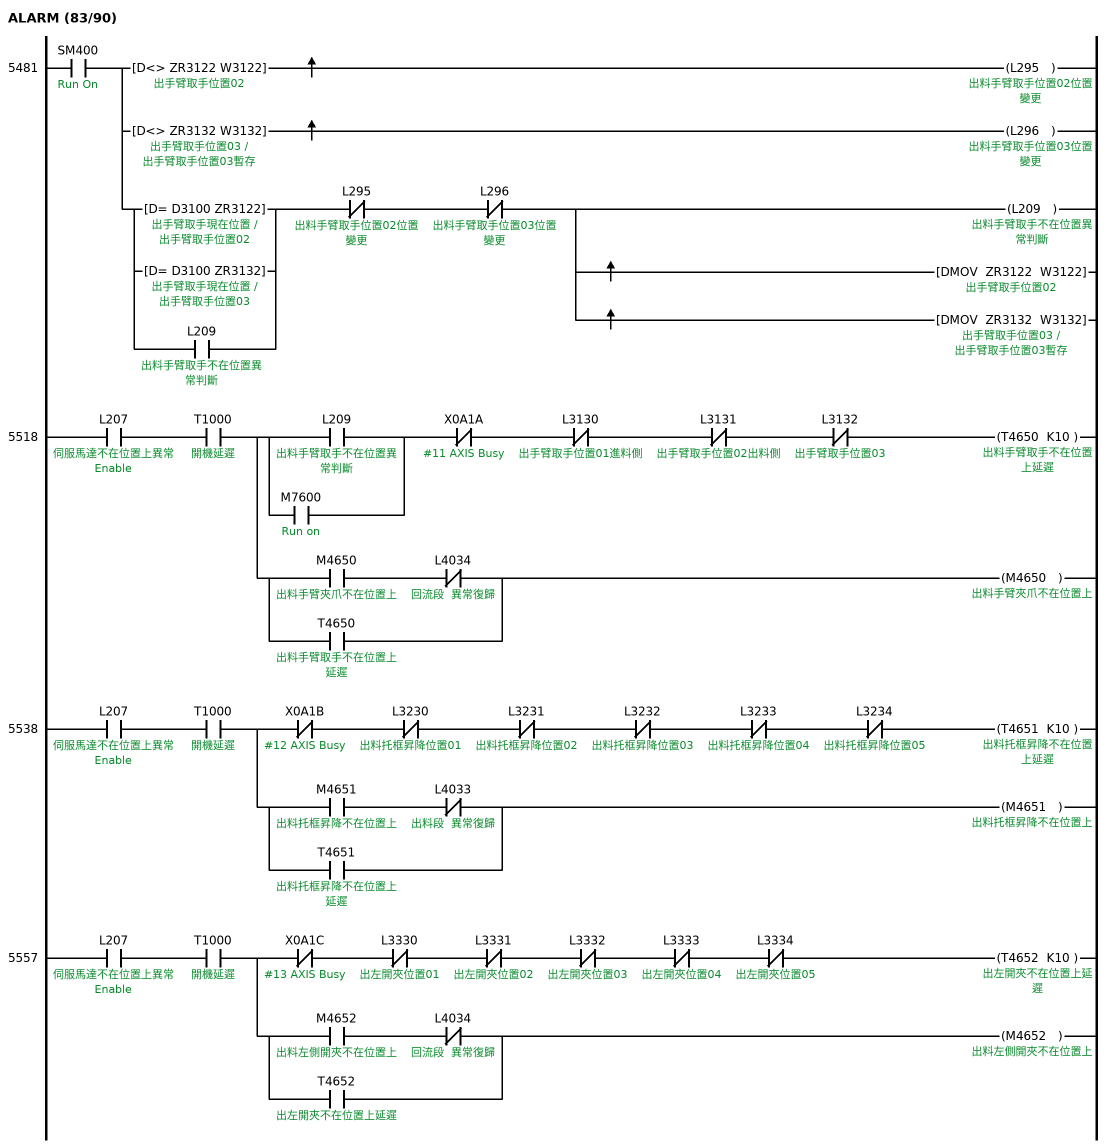
5481  LD      SM400  ; Run On
      MPS
      ANDD<>  ZR3122 W3122  ; 出手臂取手位置02
      MEP
      OUT     L295  ; 出料手臂取手位置02位置變更
      MRD
      ANDD<>  ZR3132 W3132  ; 出手臂取手位置03 / 出手臂取手位置03暫存
      MEP
      OUT     L296  ; 出料手臂取手位置03位置變更
      MPP
      LDD=    D3100 ZR3122  ; 出手臂取手現在位置 / 出手臂取手位置02
      ORD=    D3100 ZR3132  ; 出手臂取手現在位置 / 出手臂取手位置03
      OR      L209  ; 出料手臂取手不在位置異常判斷
      ANB
      ANI     L295  ; 出料手臂取手位置02位置變更
      ANI     L296  ; 出料手臂取手位置03位置變更
      OUT     L209  ; 出料手臂取手不在位置異常判斷
      MPS
      MEP
      DMOV    ZR3122 W3122
      MPP
      MEP
      DMOV    ZR3132 W3132
5518  LD      L207  ; 伺服馬達不在位置上異常  Enable
      AND     T1000  ; 開機延遲
      MPS
      LD      L209  ; 出料手臂取手不在位置異常判斷
      OR      M7600  ; Run on
      ANB
      ANI     X0A1A  ; #11 AXIS Busy
      ANI     L3130  ; 出手臂取手位置01進料側
      ANI     L3131  ; 出手臂取手位置02出料側
      ANI     L3132  ; 出手臂取手位置03
      OUT     T4650 K10  ; 出料手臂取手不在位置上延遲
      MPP
      LD      M4650  ; 出料手臂夾爪不在位置上
      ANI     L4034  ; 回流段  異常復歸
      OR      T4650  ; 出料手臂取手不在位置上延遲
      ANB
      OUT     M4650  ; 出料手臂夾爪不在位置上
5538  LD      L207  ; 伺服馬達不在位置上異常  Enable
      AND     T1000  ; 開機延遲
      MPS
      ANI     X0A1B  ; #12 AXIS Busy
      ANI     L3230  ; 出料托框昇降位置01
      ANI     L3231  ; 出料托框昇降位置02
      ANI     L3232  ; 出料托框昇降位置03
      ANI     L3233  ; 出料托框昇降位置04
      ANI     L3234  ; 出料托框昇降位置05
      OUT     T4651 K10  ; 出料托框昇降不在位置上延遲
      MPP
      LD      M4651  ; 出料托框昇降不在位置上
      ANI     L4033  ; 出料段  異常復歸
      OR      T4651  ; 出料托框昇降不在位置上延遲
      ANB
      OUT     M4651  ; 出料托框昇降不在位置上
5557  LD      L207  ; 伺服馬達不在位置上異常  Enable
      AND     T1000  ; 開機延遲
      MPS
      ANI     X0A1C  ; #13 AXIS Busy
      ANI     L3330  ; 出左開夾位置01
      ANI     L3331  ; 出左開夾位置02
      ANI     L3332  ; 出左開夾位置03
      ANI     L3333  ; 出左開夾位置04
      ANI     L3334  ; 出左開夾位置05
      OUT     T4652 K10  ; 出左開夾不在位置上延遲
      MPP
      LD      M4652  ; 出料左側開夾不在位置上
      ANI     L4034  ; 回流段  異常復歸
      OR      T4652  ; 出左開夾不在位置上延遲
      ANB
      OUT     M4652  ; 出料左側開夾不在位置上
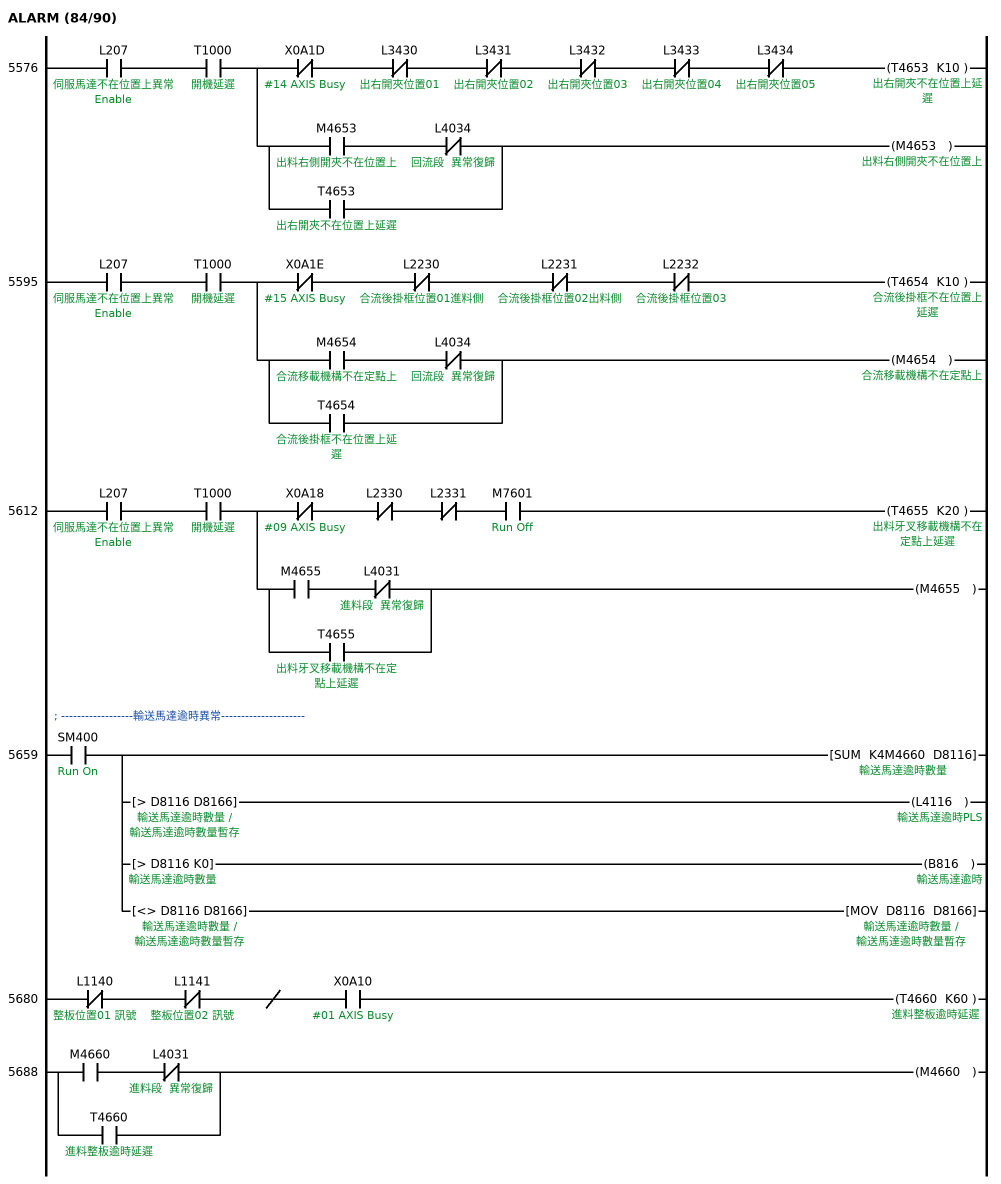
5576  LD      L207  ; 伺服馬達不在位置上異常  Enable
      AND     T1000  ; 開機延遲
      MPS
      ANI     X0A1D  ; #14 AXIS Busy
      ANI     L3430  ; 出右開夾位置01
      ANI     L3431  ; 出右開夾位置02
      ANI     L3432  ; 出右開夾位置03
      ANI     L3433  ; 出右開夾位置04
      ANI     L3434  ; 出右開夾位置05
      OUT     T4653 K10  ; 出右開夾不在位置上延遲
      MPP
      LD      M4653  ; 出料右側開夾不在位置上
      ANI     L4034  ; 回流段  異常復歸
      OR      T4653  ; 出右開夾不在位置上延遲
      ANB
      OUT     M4653  ; 出料右側開夾不在位置上
5595  LD      L207  ; 伺服馬達不在位置上異常  Enable
      AND     T1000  ; 開機延遲
      MPS
      ANI     X0A1E  ; #15 AXIS Busy
      ANI     L2230  ; 合流後掛框位置01進料側
      ANI     L2231  ; 合流後掛框位置02出料側
      ANI     L2232  ; 合流後掛框位置03
      OUT     T4654 K10  ; 合流後掛框不在位置上延遲
      MPP
      LD      M4654  ; 合流移載機構不在定點上
      ANI     L4034  ; 回流段  異常復歸
      OR      T4654  ; 合流後掛框不在位置上延遲
      ANB
      OUT     M4654  ; 合流移載機構不在定點上
5612  LD      L207  ; 伺服馬達不在位置上異常  Enable
      AND     T1000  ; 開機延遲
      MPS
      ANI     X0A18  ; #09 AXIS Busy
      ANI     L2330
      ANI     L2331
      AND     M7601  ; Run Off
      OUT     T4655 K20  ; 出料牙叉移載機構不在定點上延遲
      MPP
      LD      M4655
      ANI     L4031  ; 進料段  異常復歸
      OR      T4655  ; 出料牙叉移載機構不在定點上延遲
      ANB
      OUT     M4655
; ------------------輸送馬達逾時異常---------------------
5659  LD      SM400  ; Run On
      SUM     K4M4660 D8116  ; 輸送馬達逾時數量
      MPS
      AND>    D8116 D8166  ; 輸送馬達逾時數量 / 輸送馬達逾時數量暫存
      OUT     L4116  ; 輸送馬達逾時PLS
      MRD
      AND>    D8116 K0  ; 輸送馬達逾時數量
      OUT     B816  ; 輸送馬達逾時
      MPP
      AND<>   D8116 D8166  ; 輸送馬達逾時數量 / 輸送馬達逾時數量暫存
      MOV     D8116 D8166
5680  LDI     L1140  ; 整板位置01 訊號
      ANI     L1141  ; 整板位置02 訊號
      INV
      AND     X0A10  ; #01 AXIS Busy
      OUT     T4660 K60  ; 進料整板逾時延遲
5688  LD      M4660
      ANI     L4031  ; 進料段  異常復歸
      OR      T4660  ; 進料整板逾時延遲
      OUT     M4660
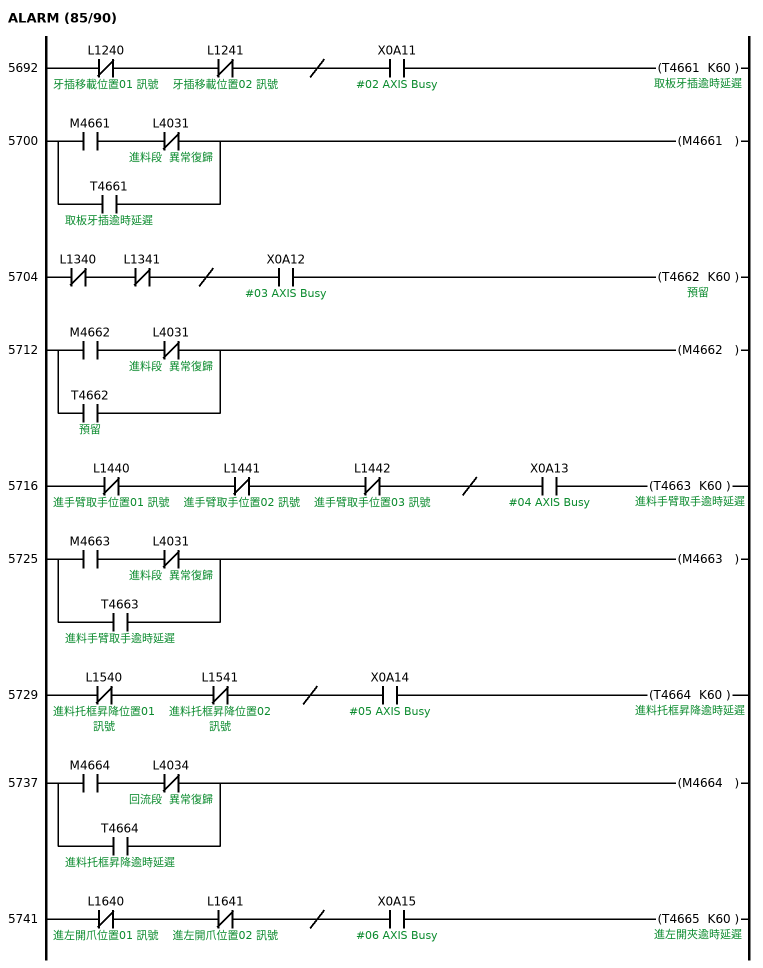
5692  LDI     L1240  ; 牙插移載位置01 訊號
      ANI     L1241  ; 牙插移載位置02 訊號
      INV
      AND     X0A11  ; #02 AXIS Busy
      OUT     T4661 K60  ; 取板牙插逾時延遲
5700  LD      M4661
      ANI     L4031  ; 進料段  異常復歸
      OR      T4661  ; 取板牙插逾時延遲
      OUT     M4661
5704  LDI     L1340
      ANI     L1341
      INV
      AND     X0A12  ; #03 AXIS Busy
      OUT     T4662 K60  ; 預留
5712  LD      M4662
      ANI     L4031  ; 進料段  異常復歸
      OR      T4662  ; 預留
      OUT     M4662
5716  LDI     L1440  ; 進手臂取手位置01 訊號
      ANI     L1441  ; 進手臂取手位置02 訊號
      ANI     L1442  ; 進手臂取手位置03 訊號
      INV
      AND     X0A13  ; #04 AXIS Busy
      OUT     T4663 K60  ; 進料手臂取手逾時延遲
5725  LD      M4663
      ANI     L4031  ; 進料段  異常復歸
      OR      T4663  ; 進料手臂取手逾時延遲
      OUT     M4663
5729  LDI     L1540  ; 進料托框昇降位置01 訊號
      ANI     L1541  ; 進料托框昇降位置02 訊號
      INV
      AND     X0A14  ; #05 AXIS Busy
      OUT     T4664 K60  ; 進料托框昇降逾時延遲
5737  LD      M4664
      ANI     L4034  ; 回流段  異常復歸
      OR      T4664  ; 進料托框昇降逾時延遲
      OUT     M4664
5741  LDI     L1640  ; 進左開爪位置01 訊號
      ANI     L1641  ; 進左開爪位置02 訊號
      INV
      AND     X0A15  ; #06 AXIS Busy
      OUT     T4665 K60  ; 進左開夾逾時延遲
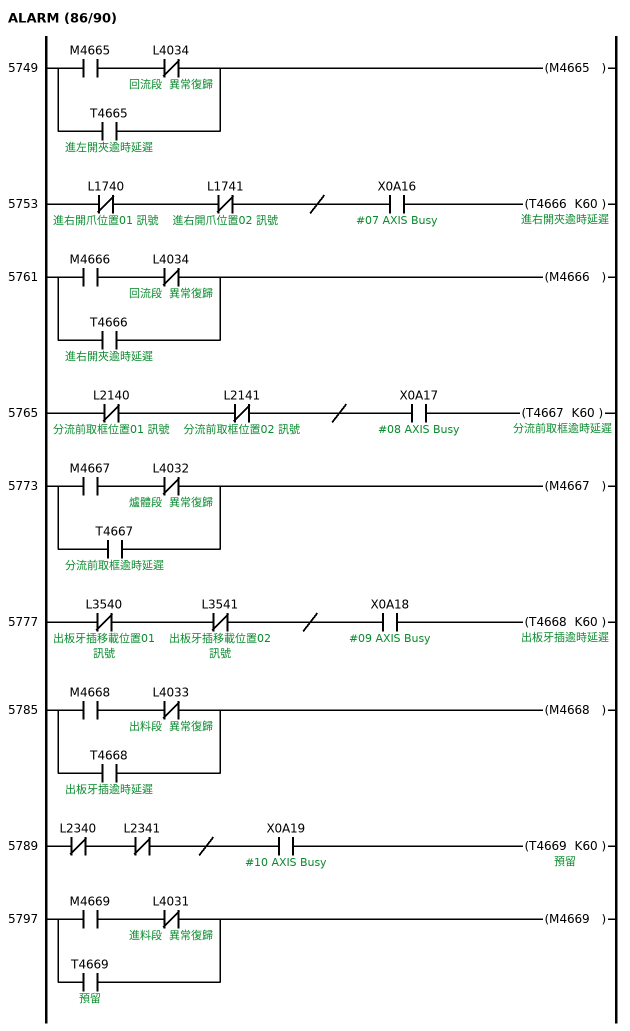
5749  LD      M4665
      ANI     L4034  ; 回流段  異常復歸
      OR      T4665  ; 進左開夾逾時延遲
      OUT     M4665
5753  LDI     L1740  ; 進右開爪位置01 訊號
      ANI     L1741  ; 進右開爪位置02 訊號
      INV
      AND     X0A16  ; #07 AXIS Busy
      OUT     T4666 K60  ; 進右開夾逾時延遲
5761  LD      M4666
      ANI     L4034  ; 回流段  異常復歸
      OR      T4666  ; 進右開夾逾時延遲
      OUT     M4666
5765  LDI     L2140  ; 分流前取框位置01 訊號
      ANI     L2141  ; 分流前取框位置02 訊號
      INV
      AND     X0A17  ; #08 AXIS Busy
      OUT     T4667 K60  ; 分流前取框逾時延遲
5773  LD      M4667
      ANI     L4032  ; 爐體段  異常復歸
      OR      T4667  ; 分流前取框逾時延遲
      OUT     M4667
5777  LDI     L3540  ; 出板牙插移載位置01 訊號
      ANI     L3541  ; 出板牙插移載位置02 訊號
      INV
      AND     X0A18  ; #09 AXIS Busy
      OUT     T4668 K60  ; 出板牙插逾時延遲
5785  LD      M4668
      ANI     L4033  ; 出料段  異常復歸
      OR      T4668  ; 出板牙插逾時延遲
      OUT     M4668
5789  LDI     L2340
      ANI     L2341
      INV
      AND     X0A19  ; #10 AXIS Busy
      OUT     T4669 K60  ; 預留
5797  LD      M4669
      ANI     L4031  ; 進料段  異常復歸
      OR      T4669  ; 預留
      OUT     M4669
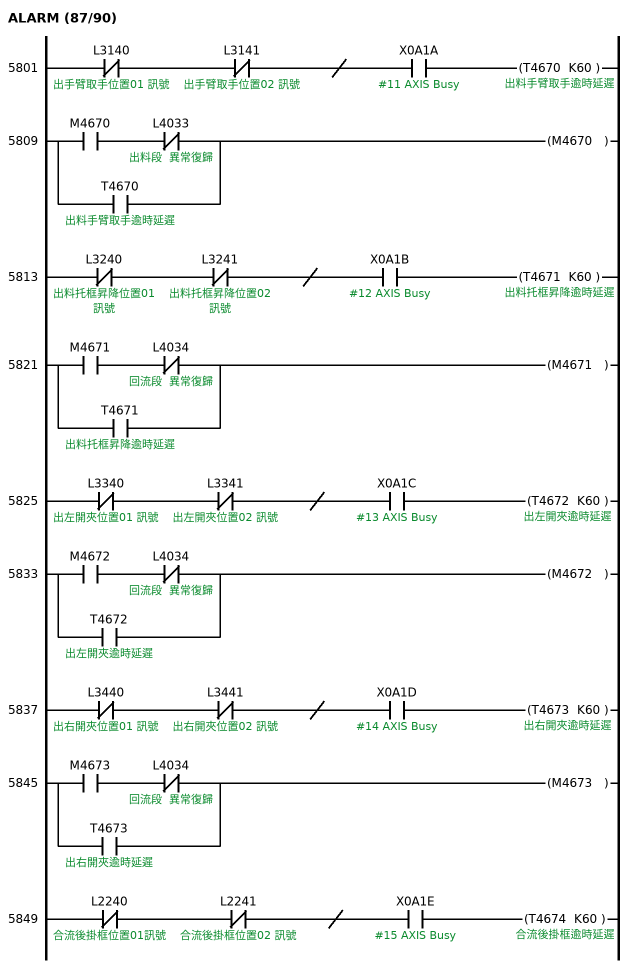
5801  LDI     L3140  ; 出手臂取手位置01 訊號
      ANI     L3141  ; 出手臂取手位置02 訊號
      INV
      AND     X0A1A  ; #11 AXIS Busy
      OUT     T4670 K60  ; 出料手臂取手逾時延遲
5809  LD      M4670
      ANI     L4033  ; 出料段  異常復歸
      OR      T4670  ; 出料手臂取手逾時延遲
      OUT     M4670
5813  LDI     L3240  ; 出料托框昇降位置01 訊號
      ANI     L3241  ; 出料托框昇降位置02 訊號
      INV
      AND     X0A1B  ; #12 AXIS Busy
      OUT     T4671 K60  ; 出料托框昇降逾時延遲
5821  LD      M4671
      ANI     L4034  ; 回流段  異常復歸
      OR      T4671  ; 出料托框昇降逾時延遲
      OUT     M4671
5825  LDI     L3340  ; 出左開夾位置01 訊號
      ANI     L3341  ; 出左開夾位置02 訊號
      INV
      AND     X0A1C  ; #13 AXIS Busy
      OUT     T4672 K60  ; 出左開夾逾時延遲
5833  LD      M4672
      ANI     L4034  ; 回流段  異常復歸
      OR      T4672  ; 出左開夾逾時延遲
      OUT     M4672
5837  LDI     L3440  ; 出右開夾位置01 訊號
      ANI     L3441  ; 出右開夾位置02 訊號
      INV
      AND     X0A1D  ; #14 AXIS Busy
      OUT     T4673 K60  ; 出右開夾逾時延遲
5845  LD      M4673
      ANI     L4034  ; 回流段  異常復歸
      OR      T4673  ; 出右開夾逾時延遲
      OUT     M4673
5849  LDI     L2240  ; 合流後掛框位置01訊號
      ANI     L2241  ; 合流後掛框位置02 訊號
      INV
      AND     X0A1E  ; #15 AXIS Busy
      OUT     T4674 K60  ; 合流後掛框逾時延遲
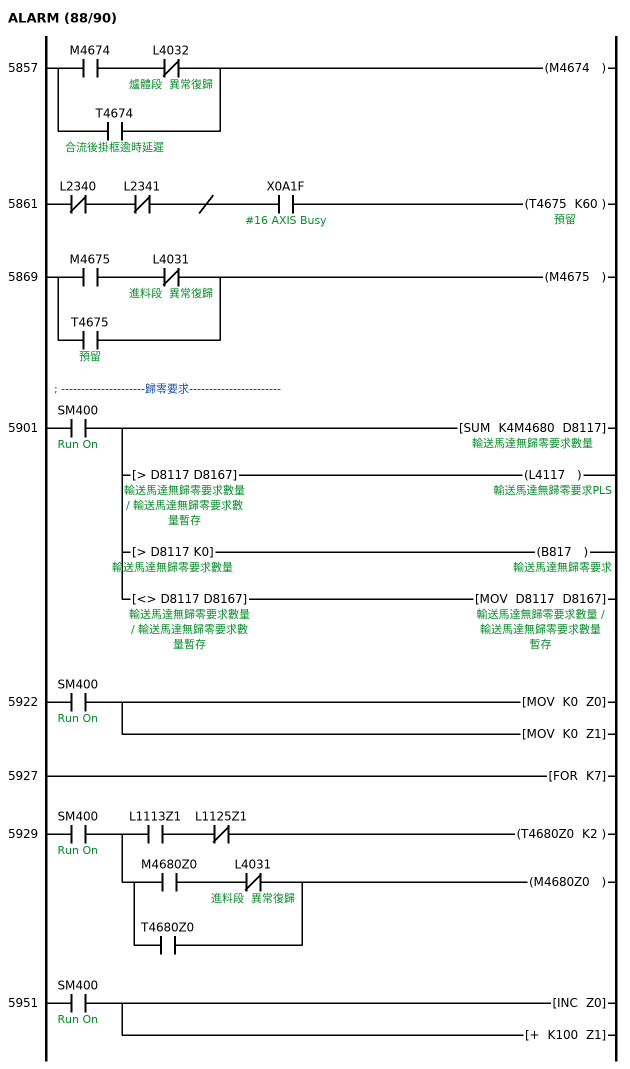
5857  LD      M4674
      ANI     L4032  ; 爐體段  異常復歸
      OR      T4674  ; 合流後掛框逾時延遲
      OUT     M4674
5861  LDI     L2340
      ANI     L2341
      INV
      AND     X0A1F  ; #16 AXIS Busy
      OUT     T4675 K60  ; 預留
5869  LD      M4675
      ANI     L4031  ; 進料段  異常復歸
      OR      T4675  ; 預留
      OUT     M4675
; ---------------------歸零要求-----------------------
5901  LD      SM400  ; Run On
      SUM     K4M4680 D8117  ; 進料整板歸零要求異常 / 輸送馬達無歸零要求數量
      MPS
      AND>    D8117 D8167  ; 輸送馬達無歸零要求數量 / 輸送馬達無歸零要求數量暫存
      OUT     L4117  ; 輸送馬達無歸零要求PLS
      MRD
      AND>    D8117 K0  ; 輸送馬達無歸零要求數量
      OUT     B817  ; 輸送馬達無歸零要求
      MPP
      AND<>   D8117 D8167  ; 輸送馬達無歸零要求數量 / 輸送馬達無歸零要求數量暫存
      MOV     D8117 D8167
5922  LD      SM400  ; Run On
      MOV     K0 Z0
      MOV     K0 Z1
5927  FOR     K7
5929  LD      SM400  ; Run On
      MPS
      AND     L1113Z1
      ANI     L1125Z1
      OUT     T4680Z0 K2
      MPP
      LD      M4680Z0
      ANI     L4031  ; 進料段  異常復歸
      OR      T4680Z0
      ANB
      OUT     M4680Z0
5951  LD      SM400  ; Run On
      INC     Z0
      +       K100 Z1
